TYPE DustIQ_Standard :
STRUCT
	MesData : DustIQ ; (* Child struct  *)
END_STRUCT
END_TYPE

(* stored: Version 1.1.0.1, ProductVersion 3.1.4024.11
   DUT DustIQ_Standard: Id {914987ba-2f4e-4000-85de-206365152723} *)
